FUNCTION_BLOCK ABSTRACT FBA_Drive IMPLEMENTS I_Drive
VAR_INPUT
	bEnable : BOOL;
END_VAR
VAR //constructor
	limitSensorDefaultState : BOOL;
	//when a traverse sensor is opposite of this value, the respective property becomes TRUE
	//all sensors for a drive should be of the same type - do not mix & match PNP and NPN sensors on the same drive
END_VAR
VAR		
	homingComplete : BOOL;
	step : Homing;
	
	innerLimit AT %I* : BOOL; //replacable with homeLimit
	home AT %I* : BOOL;
	//not all drives have a rear limit, drives that do must extend from FBA_TrifectaDrive
END_VAR
(*
this abstract FB only specifies the minimum data for any drive
*)

{attribute 'monitoring':='call'}
PROPERTY ABSTRACT Active : BOOL
GET
END_GET
END_PROPERTY

{attribute 'monitoring':='call'}
PROPERTY AtHome : BOOL
GET
AtHome := home <> limitSensorDefaultState;
END_GET
END_PROPERTY

{attribute 'monitoring':='call'}
PROPERTY AtInnerLimit : BOOL
GET
AtInnerLimit := innerLimit <> limitSensorDefaultState;
END_GET
END_PROPERTY

{attribute 'monitoring':='call'}
PROPERTY ABSTRACT Error : BOOL
GET
END_GET
END_PROPERTY

{attribute 'monitoring':='call'}
PROPERTY HomeSet : BOOL
GET
HomeSet := homingComplete;
END_GET
END_PROPERTY

{attribute 'TcRpcEnable'}
METHOD ABSTRACT homingSequence : BOOL
VAR_INPUT
END_VAR
END_METHOD

{attribute 'TcRpcEnable'}
METHOD ABSTRACT reset : BOOL
VAR_INPUT
END_VAR
END_METHOD

{attribute 'TcRpcEnable'}
METHOD ABSTRACT stop : BOOL
VAR_INPUT
END_VAR
END_METHOD

METHOD ABSTRACT toHome : BOOL
VAR_INPUT
END_VAR
END_METHOD

END_FUNCTION_BLOCK

(* stored: Version 1.1.0.1, ProductVersion 3.1.4024.11
   POU FBA_Drive: Id {2de1cb23-32f2-4219-89c5-fb81e366fa09}, SpecialFunc None
   Folder Abstract: Id {c5aa1f87-afe2-4e7f-ace1-de8c3966dd88}
   Folder Complete: Id {0b25e528-0c48-465e-93f4-3e9dd063fa23}
   Property Active: Id {d1381e43-e73a-47e2-a25c-0a860678c4a2}
   Get Get: Id {5e5510a3-652b-4cb8-aa27-d7e65ef261f6}
   Property AtHome: Id {5b35509c-86aa-4d7c-afa4-3c87c4fd2400}
   Get Get: Id {0fdc76c7-f6c5-49ce-8b43-d9df2ab87af9}
   Property AtInnerLimit: Id {71d3a6c6-612d-4635-b770-694d48510893}
   Get Get: Id {c5322a12-e6cf-430c-9246-e85c68be0e69}
   Property Error: Id {f91f2d47-7f8e-4d3d-9a9c-df891ddd96e0}
   Get Get: Id {cf5a7583-df79-4b7c-9e12-e919740dc30d}
   Property HomeSet: Id {6a9a7f84-8a36-4778-a429-3d940b40bc6e}
   Get Get: Id {32b7fd94-22c6-4de0-91cb-7302016f9e27}
   Method homingSequence: Id {7135e606-2f38-4ced-9625-cc9303ca45bf}
   Method reset: Id {89936125-0d83-4e3e-88d4-6abae24e37b7}
   Method stop: Id {b225f2f1-2348-4f1a-aec3-8bf30e5b2053}
   Method toHome: Id {efe7f4e0-a6c1-4d7d-9b20-2517bed59931} *)
